// TIA Portal V19 export
FUNCTION_BLOCK "FESTO_CMMT_ST"   // FB4, LAD
{ S7_Optimized_Access := 'TRUE' }
// stored: MemoryReserve 100, SetENOAutomatically false
   VAR
      Festo_PtP_Drives_PN_Instance { S7_SetPoint := 'True'} : "Festo_PtP_Drives_PN";
   END_VAR
   VAR_TEMP
      i : Int;
   END_VAR
BEGIN

REGION Network 1
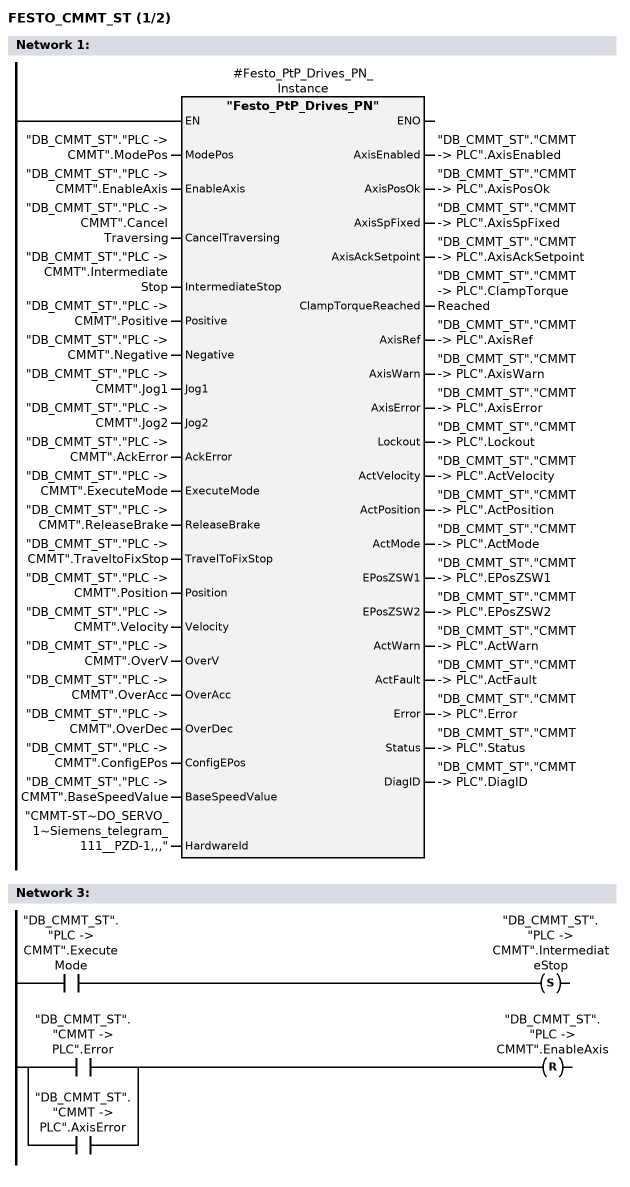
   RUNG wire#powerrail
      #Festo_PtP_Drives_PN_Instance(ModePos := "DB_CMMT_ST"."PLC -> CMMT".ModePos, EnableAxis := "DB_CMMT_ST"."PLC -> CMMT".EnableAxis, CancelTraversing := "DB_CMMT_ST"."PLC -> CMMT".CancelTraversing, IntermediateStop := "DB_CMMT_ST"."PLC -> CMMT".IntermediateStop, Positive := "DB_CMMT_ST"."PLC -> CMMT".Positive, Negative := "DB_CMMT_ST"."PLC -> CMMT".Negative, Jog1 := "DB_CMMT_ST"."PLC -> CMMT".Jog1, Jog2 := "DB_CMMT_ST"."PLC -> CMMT".Jog2, AckError := "DB_CMMT_ST"."PLC -> CMMT".AckError, ExecuteMode := "DB_CMMT_ST"."PLC -> CMMT".ExecuteMode, ReleaseBrake := "DB_CMMT_ST"."PLC -> CMMT".ReleaseBrake, TravelToFixStop := "DB_CMMT_ST"."PLC -> CMMT".TraveltoFixStop, Position := "DB_CMMT_ST"."PLC -> CMMT".Position, Velocity := "DB_CMMT_ST"."PLC -> CMMT".Velocity, OverV := "DB_CMMT_ST"."PLC -> CMMT".OverV, OverAcc := "DB_CMMT_ST"."PLC -> CMMT".OverAcc, OverDec := "DB_CMMT_ST"."PLC -> CMMT".OverDec, ConfigEPos := "DB_CMMT_ST"."PLC -> CMMT".ConfigEPos, BaseSpeedValue := "DB_CMMT_ST"."PLC -> CMMT".BaseSpeedValue, HardwareId := "CMMT-ST~DO_SERVO_1~Siemens_telegram_111__PZD-1,,,", AxisEnabled => "DB_CMMT_ST"."CMMT -> PLC".AxisEnabled, AxisPosOk => "DB_CMMT_ST"."CMMT -> PLC".AxisPosOk, AxisSpFixed => "DB_CMMT_ST"."CMMT -> PLC".AxisSpFixed, AxisAckSetpoint => "DB_CMMT_ST"."CMMT -> PLC".AxisAckSetpoint, ClampTorqueReached => "DB_CMMT_ST"."CMMT -> PLC".ClampTorqueReached, AxisRef => "DB_CMMT_ST"."CMMT -> PLC".AxisRef, AxisWarn => "DB_CMMT_ST"."CMMT -> PLC".AxisWarn, AxisError => "DB_CMMT_ST"."CMMT -> PLC".AxisError, Lockout => "DB_CMMT_ST"."CMMT -> PLC".Lockout, ActVelocity => "DB_CMMT_ST"."CMMT -> PLC".ActVelocity, ActPosition => "DB_CMMT_ST"."CMMT -> PLC".ActPosition, ActMode => "DB_CMMT_ST"."CMMT -> PLC".ActMode, EPosZSW1 => "DB_CMMT_ST"."CMMT -> PLC".EPosZSW1, EPosZSW2 => "DB_CMMT_ST"."CMMT -> PLC".EPosZSW2, ActWarn => "DB_CMMT_ST"."CMMT -> PLC".ActWarn, ActFault => "DB_CMMT_ST"."CMMT -> PLC".ActFault, Error => "DB_CMMT_ST"."CMMT -> PLC".Error, Status => "DB_CMMT_ST"."CMMT -> PLC".Status, DiagID => "DB_CMMT_ST"."CMMT -> PLC".DiagID)
   END_RUNG
   // the same network as SCL:
   #Festo_PtP_Drives_PN_Instance(ModePos := "DB_CMMT_ST"."PLC -> CMMT".ModePos,   // "Festo_PtP_Drives_PN"
                           EnableAxis := "DB_CMMT_ST"."PLC -> CMMT".EnableAxis,
                           CancelTraversing := "DB_CMMT_ST"."PLC -> CMMT".CancelTraversing,
                           IntermediateStop := "DB_CMMT_ST"."PLC -> CMMT".IntermediateStop,
                           Positive := "DB_CMMT_ST"."PLC -> CMMT".Positive,
                           Negative := "DB_CMMT_ST"."PLC -> CMMT".Negative,
                           Jog1 := "DB_CMMT_ST"."PLC -> CMMT".Jog1,
                           Jog2 := "DB_CMMT_ST"."PLC -> CMMT".Jog2,
                           AckError := "DB_CMMT_ST"."PLC -> CMMT".AckError,
                           ExecuteMode := "DB_CMMT_ST"."PLC -> CMMT".ExecuteMode,
                           ReleaseBrake := "DB_CMMT_ST"."PLC -> CMMT".ReleaseBrake,
                           TravelToFixStop := "DB_CMMT_ST"."PLC -> CMMT".TraveltoFixStop,
                           Position := "DB_CMMT_ST"."PLC -> CMMT".Position,
                           Velocity := "DB_CMMT_ST"."PLC -> CMMT".Velocity,
                           OverV := "DB_CMMT_ST"."PLC -> CMMT".OverV,
                           OverAcc := "DB_CMMT_ST"."PLC -> CMMT".OverAcc,
                           OverDec := "DB_CMMT_ST"."PLC -> CMMT".OverDec,
                           ConfigEPos := "DB_CMMT_ST"."PLC -> CMMT".ConfigEPos,
                           BaseSpeedValue := "DB_CMMT_ST"."PLC -> CMMT".BaseSpeedValue,
                           HardwareId := "CMMT-ST~DO_SERVO_1~Siemens_telegram_111__PZD-1,,,",
                           AxisEnabled => "DB_CMMT_ST"."CMMT -> PLC".AxisEnabled,
                           AxisPosOk => "DB_CMMT_ST"."CMMT -> PLC".AxisPosOk,
                           AxisSpFixed => "DB_CMMT_ST"."CMMT -> PLC".AxisSpFixed,
                           AxisAckSetpoint => "DB_CMMT_ST"."CMMT -> PLC".AxisAckSetpoint,
                           ClampTorqueReached => "DB_CMMT_ST"."CMMT -> PLC".ClampTorqueReached,
                           AxisRef => "DB_CMMT_ST"."CMMT -> PLC".AxisRef,
                           AxisWarn => "DB_CMMT_ST"."CMMT -> PLC".AxisWarn,
                           AxisError => "DB_CMMT_ST"."CMMT -> PLC".AxisError,
                           Lockout => "DB_CMMT_ST"."CMMT -> PLC".Lockout,
                           ActVelocity => "DB_CMMT_ST"."CMMT -> PLC".ActVelocity,
                           ActPosition => "DB_CMMT_ST"."CMMT -> PLC".ActPosition,
                           ActMode => "DB_CMMT_ST"."CMMT -> PLC".ActMode,
                           EPosZSW1 => "DB_CMMT_ST"."CMMT -> PLC".EPosZSW1,
                           EPosZSW2 => "DB_CMMT_ST"."CMMT -> PLC".EPosZSW2,
                           ActWarn => "DB_CMMT_ST"."CMMT -> PLC".ActWarn,
                           ActFault => "DB_CMMT_ST"."CMMT -> PLC".ActFault,
                           Error => "DB_CMMT_ST"."CMMT -> PLC".Error,
                           Status => "DB_CMMT_ST"."CMMT -> PLC".Status,
                           DiagID => "DB_CMMT_ST"."CMMT -> PLC".DiagID);
END_REGION

REGION Network 2 (SCL): Convert Veolocity and Position in mm/s and mm
   REGION Convert Setposition from mm TO 1000_Unit
       "DB_CMMT_ST"."PLC -> CMMT".Position   := REAL_TO_DINT("DB_CMMT_ST".SetPosition_mm * 1000.0);
       "DB_CMMT_ST".HMI.Scaled_SetpointPosition := "DB_CMMT_ST".SetPosition_mm / 150.0;
   END_REGION

   REGION Convert Setvelocity 
       "DB_CMMT_ST"."PLC -> CMMT".Velocity := REAL_TO_DINT("DB_CMMT_ST".SetVelocity_mm_s);
   END_REGION

   REGION Convert Actual Position from 1000Unit to mm
       "DB_CMMT_ST".ActualPos_mm := "DB_CMMT_ST"."CMMT -> PLC".ActPosition / 1000.0;
       // Scale actual position for HMI
       "DB_CMMT_ST".HMI.Scaled_ActualPos := "DB_CMMT_ST".ActualPos_mm / 100; // Value in cm
   END_REGION

   REGION Convert Actual velocity from 1000Unit TO mm/s
       "DB_CMMT_ST".AcutalVelocity_mm_s := "DB_CMMT_ST"."CMMT -> PLC".ActVelocity * 1000.0;
   END_REGION
END_REGION

REGION Network 3
   RUNG wire#powerrail
      Contact( "DB_CMMT_ST"."PLC -> CMMT".ExecuteMode )
      S_Coil( "DB_CMMT_ST"."PLC -> CMMT".IntermediateStop )
   END_RUNG
   RUNG wire#powerrail
      Contact( "DB_CMMT_ST"."CMMT -> PLC".Error )
      wire#w1
      R_Coil( "DB_CMMT_ST"."PLC -> CMMT".EnableAxis )
   END_RUNG
   RUNG wire#powerrail
      Contact( "DB_CMMT_ST"."CMMT -> PLC".AxisError )
   END_RUNG wire#w1
   // the same network as SCL:
   IF "DB_CMMT_ST"."PLC -> CMMT".ExecuteMode THEN
       "DB_CMMT_ST"."PLC -> CMMT".IntermediateStop := TRUE;
   END_IF;
   IF "DB_CMMT_ST"."CMMT -> PLC".Error OR "DB_CMMT_ST"."CMMT -> PLC".AxisError THEN
       "DB_CMMT_ST"."PLC -> CMMT".EnableAxis := FALSE;
   END_IF;
END_REGION

REGION Network 4: Festo Calmping Torque
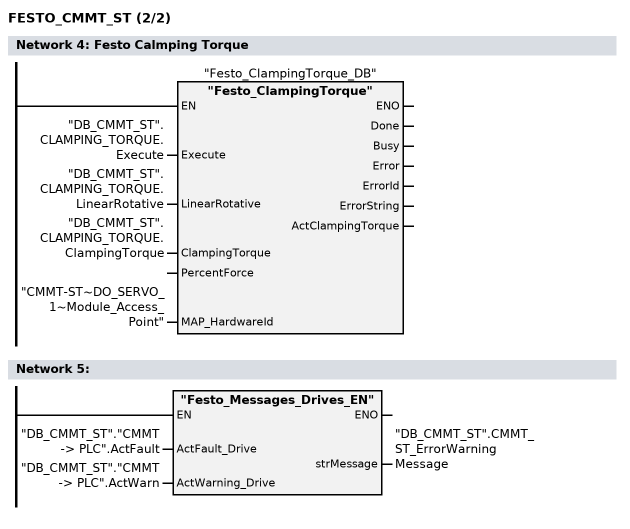
   RUNG wire#powerrail
      "Festo_ClampingTorque_DB"(Execute := "DB_CMMT_ST".CLAMPING_TORQUE.Execute, LinearRotative := "DB_CMMT_ST".CLAMPING_TORQUE.LinearRotative, ClampingTorque := "DB_CMMT_ST".CLAMPING_TORQUE.ClampingTorque, PercentForce :=, MAP_HardwareId := "CMMT-ST~DO_SERVO_1~Module_Access_Point", Done =>, Busy =>, Error =>, ErrorId =>, ErrorString =>, ActClampingTorque =>)
   END_RUNG
   // the same network as SCL:
   "Festo_ClampingTorque_DB"(Execute := "DB_CMMT_ST".CLAMPING_TORQUE.Execute,   // "Festo_ClampingTorque"
                           LinearRotative := "DB_CMMT_ST".CLAMPING_TORQUE.LinearRotative,
                           ClampingTorque := "DB_CMMT_ST".CLAMPING_TORQUE.ClampingTorque,
                           MAP_HardwareId := "CMMT-ST~DO_SERVO_1~Module_Access_Point");
END_REGION

REGION Network 5
   RUNG wire#powerrail
      "Festo_Messages_Drives_EN"(ActFault_Drive := "DB_CMMT_ST"."CMMT -> PLC".ActFault, ActWarning_Drive := "DB_CMMT_ST"."CMMT -> PLC".ActWarn, strMessage => "DB_CMMT_ST".CMMT_ST_ErrorWarningMessage)
   END_RUNG
   // the same network as SCL:
   "Festo_Messages_Drives_EN"(ActFault_Drive := "DB_CMMT_ST"."CMMT -> PLC".ActFault,
                           ActWarning_Drive := "DB_CMMT_ST"."CMMT -> PLC".ActWarn,
                           strMessage => "DB_CMMT_ST".CMMT_ST_ErrorWarningMessage);
END_REGION
END_FUNCTION_BLOCK
